(* CoDeSys 2.3 export: ENUM_CAN.EXP *)

(* Data type in 20_CAN *)
TYPE enum_Can :
	(
		CAN_RESET_STOP		:= 0,
		CAN_RESET_START	:= 1,
		CAN_RESET_WAIT		:= 2
	);
END_TYPE
